// TIA Portal project "SocketConnection_Active" (V15.1)

(* hardware
DEVICE "S71500/ET200MP station_1"  S7-1500 station
   slot 0: "Rail_0"  Rack  6ES7 590-1***0-0AA0
   slot 1: "PLC_1"  CPU 1516-3 PN/DP  6ES7 516-3AN00-0AB0  V1.8
      slot 3: "CPU display_1"  6ES7591-1BA00-0AA0
DEVICE "S7-1200 station_1"  S7-1200 Station
   slot 0: "Rack_0"  S7-1200 Rack  Rack  V1.0
   slot 1: "PLC_2"  CPU 1212FC DC/DC/DC  6ES7 212-1AF40-0XB0  V4.2
*)

// ===== PLC "PLC_1"  CPU 1516-3 PN/DP =====

VAR_GLOBAL   // PLC tag table "Default tag table"
   "TCON_REQ" AT %M0.0 : Bool;
   "TSEND_REQ" AT %M0.1 : Bool;
   "Tag_3" AT %M0.2 : Bool;
   "Tag_4" AT %M0.3 : Bool;
   "TCON_DONE" AT %M0.4 : Bool;
   "TCON_BUSY" AT %M0.5 : Bool;
   "TCON_ERROR" AT %M0.6 : Bool;
   "TSEND_DONE" AT %M1.0 : Bool;
   "TSEND_ERROR" AT %M1.1 : Bool;
   "TSEND_BUSY" AT %M1.2 : Bool;
   "TRCV_NDR" AT %M1.3 : Bool;
   "TRCV_BUSY" AT %M1.4 : Bool;
   "TRCV_ERROR" AT %M1.5 : Bool;
   "Tag_14" AT %M1.6 : Bool;
   "TCON_DONE_PLS" AT %M1.7 : Bool;
   "TCON_DONE_COUNT" AT %MW100 : Int;
   "TSEND_DONE_PLS" AT %M2.0 : Bool;
   "TSEND_DONE_COUNT" AT %MW102 : Int;
   "Tag_19" AT %M3.1 : Bool;
   "Tag_20" AT %M5.0 : Bool;
   "Tag_21" AT %M3.3 : Bool;
   "CONNECT_RST" AT %M0.7 : Bool;
END_VAR

DATA_BLOCK "FB_TCPIP_Active_DB"   // DB6
{ S7_Optimized_Access := 'TRUE' }
VERSION : 0.1
// stored: InstanceOfName FB_TCPIP_Active
"FB_TCPIP_Active"
BEGIN
END_DATA_BLOCK

DATA_BLOCK "MyData"   // DB10
{ S7_Optimized_Access := 'FALSE' }
VERSION : 0.1
   VAR
      send_data : Array[1000..1719] of UInt;
      rcv_data : Array[0..9] of Byte;
   END_VAR
BEGIN
END_DATA_BLOCK

// folder: System blocks/Program resources

DATA_BLOCK "PLC_1_Connection_DB"   // DB2
{ S7_Optimized_Access := 'TRUE' }
AUTHOR : SIMATIC
FAMILY : MC7Plus
NAME : TC_IP_v4
VERSION : 1.0
// stored: InstanceOfName TCON_IP_v4
"TCON_IP_v4"
BEGIN
   ID := 1;
   InterfaceId := 64;
   LocalPort := 4000;
   RemotePort := 4000;
   ActiveEstablished := true;
   RemoteAddress.ADDR[1] := 192;
   RemoteAddress.ADDR[2] := 168;
   RemoteAddress.ADDR[4] := 251;
END_DATA_BLOCK

// folder: (top level)

FUNCTION_BLOCK "FB_TCPIP_Active"   // FB1, LAD
{ S7_Optimized_Access := 'TRUE' }
VERSION : 0.1
   VAR_INPUT
      REQ : Array[0..15] of Bool;
   END_VAR
   VAR
      TCON : TCON;
      TSEND : TSEND;
      TRCV : TRCV;
      TDISCON : TDISCON;
      pls : Array[0..15] of Bool;
      COUNT : Array[0..15] of Int;
   END_VAR
   VAR_TEMP   // added for the SCL form of the ladder/FBD networks
      _w1 : Bool;
      _w2 : Bool;
   END_VAR
   // // REQ[0] : TCON
   // // REQ[1] : TSEND
   // // REQ[2] : TDISCON
BEGIN

REGION Network 2: TON
END_REGION

REGION Network 3: ..Req
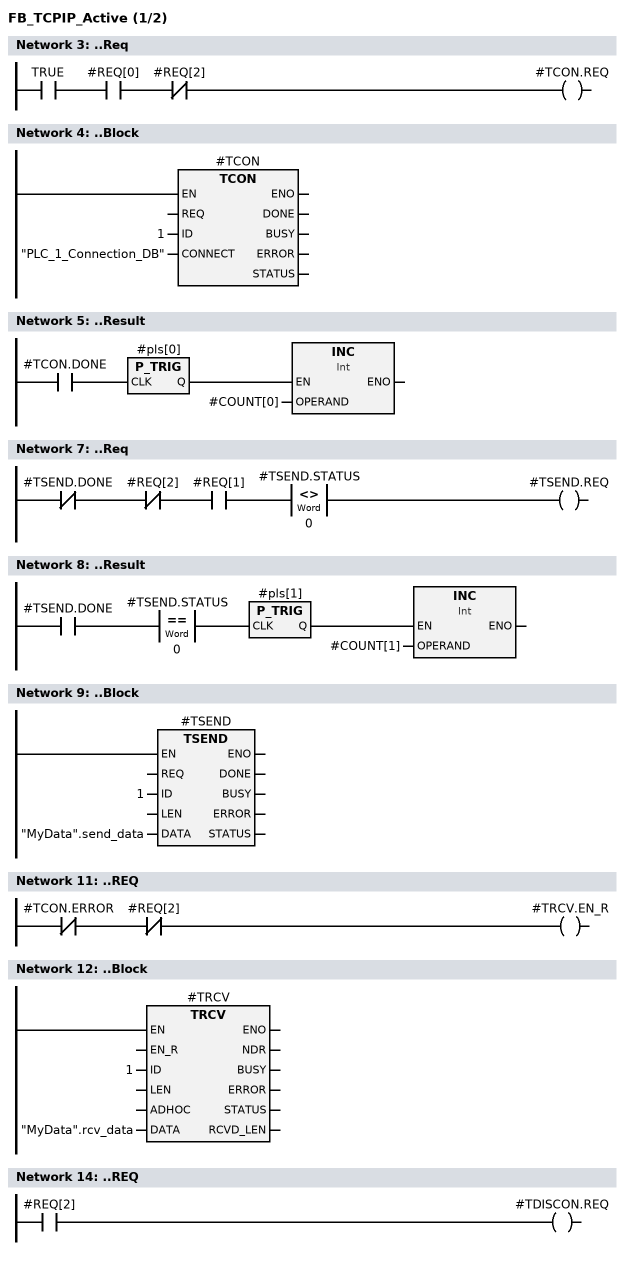
   RUNG wire#powerrail
      Contact( TRUE )
      Contact( #REQ[0] )
      I_Contact( #REQ[2] )
      Coil( #TCON.REQ )
   END_RUNG
   // the same network as SCL:
   #TCON.REQ := TRUE AND #REQ[0] AND NOT #REQ[2];
END_REGION

REGION Network 4: ..Block
   #TCON(ID := 1, CONNECT := "PLC_1_Connection_DB");   // TCON
END_REGION

REGION Network 5: ..Result
   RUNG wire#powerrail
      Contact( #TCON.DONE )
      P_Trig( #pls[0] )
      { S7_Templates := "DestType := Int" } Inc( #COUNT[0] )
   END_RUNG
   // the same network as SCL:
   #_w1 := #TCON.DONE AND NOT #pls[0];   // rising edge
   #pls[0] := #TCON.DONE;
   IF #_w1 THEN #COUNT[0] := #COUNT[0] + 1; END_IF;
END_REGION

REGION Network 6: TSEND
END_REGION

REGION Network 7: ..Req
   RUNG wire#powerrail
      I_Contact( #TSEND.DONE )
      I_Contact( #REQ[2] )
      Contact( #REQ[1] )
      { S7_Templates := "SrcType := Word" } NE_Contact(in1 := #TSEND.STATUS, in2 := 0)
      Coil( #TSEND.REQ )
   END_RUNG
   // the same network as SCL:
   #TSEND.REQ := NOT #TSEND.DONE AND NOT #REQ[2] AND #REQ[1] AND (#TSEND.STATUS <> 0);
END_REGION

REGION Network 8: ..Result
   RUNG wire#powerrail
      Contact( #TSEND.DONE )
      { S7_Templates := "SrcType := Word" } EQ_Contact(in1 := #TSEND.STATUS, in2 := 0)
      P_Trig( #pls[1] )
      { S7_Templates := "DestType := Int" } Inc( #COUNT[1] )
   END_RUNG
   // the same network as SCL:
   #_w1 := #TSEND.DONE AND (#TSEND.STATUS = 0);
   #_w2 := #_w1 AND NOT #pls[1];   // rising edge
   #pls[1] := #_w1;
   IF #_w2 THEN #COUNT[1] := #COUNT[1] + 1; END_IF;
END_REGION

REGION Network 9: ..Block
   #TSEND(ID := 1, DATA := "MyData".send_data);   // TSEND
END_REGION

REGION Network 10: TRCV
END_REGION

REGION Network 11: ..REQ
   RUNG wire#powerrail
      I_Contact( #TCON.ERROR )
      I_Contact( #REQ[2] )
      Coil( #TRCV.EN_R )
   END_RUNG
   // the same network as SCL:
   #TRCV.EN_R := NOT #TCON.ERROR AND NOT #REQ[2];
END_REGION

REGION Network 12: ..Block
   #TRCV(ID := 1, DATA := "MyData".rcv_data);   // TRCV
END_REGION

REGION Network 13: TDISCON
END_REGION

REGION Network 14: ..REQ
   RUNG wire#powerrail
      Contact( #REQ[2] )
      Coil( #TDISCON.REQ )
   END_RUNG
   // the same network as SCL:
   #TDISCON.REQ := #REQ[2];
END_REGION

REGION Network 15: ..Block
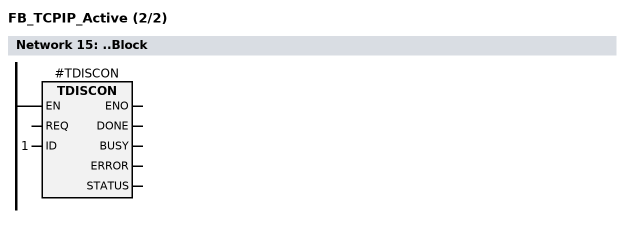
   #TDISCON(ID := 1);   // TDISCON
END_REGION
END_FUNCTION_BLOCK

FUNCTION "Backup" : Void   // FC1, LAD
{ S7_Optimized_Access := 'TRUE' }
VERSION : 0.1
   VAR_TEMP   // added for the SCL form of the ladder/FBD networks
      _w1 : Bool;
   END_VAR
BEGIN

REGION Network 2
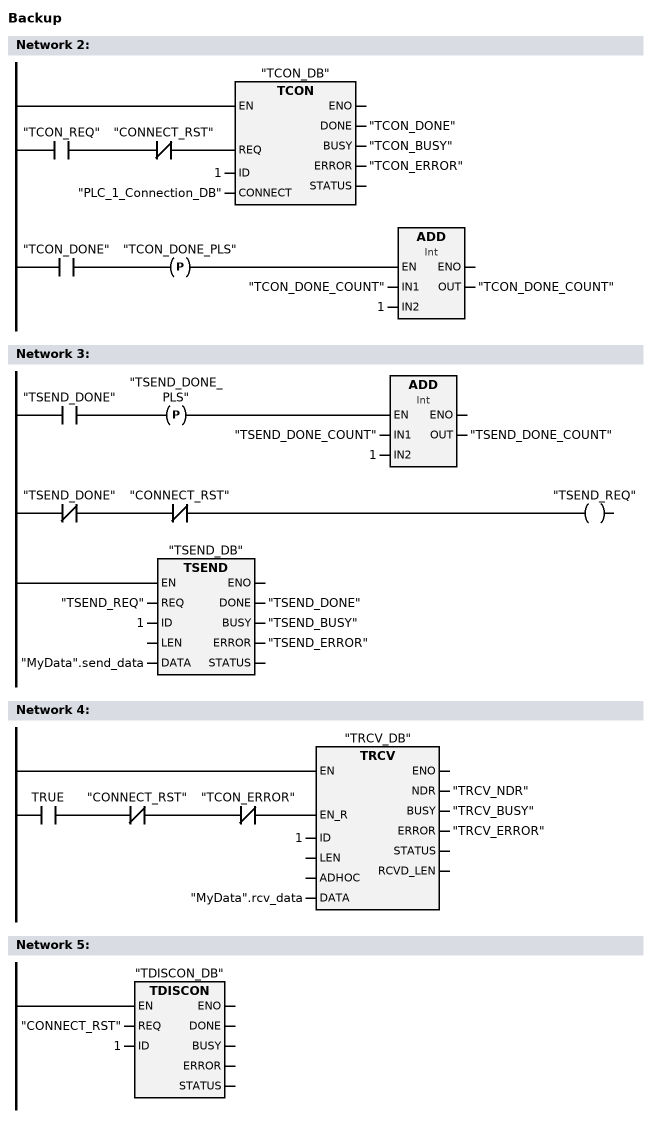
   "TCON_DB"(REQ := "TCON_REQ" AND NOT "CONNECT_RST",   // TCON
             ID := 1,
             CONNECT := "PLC_1_Connection_DB",
             DONE => "TCON_DONE",
             BUSY => "TCON_BUSY",
             ERROR => "TCON_ERROR");
   #_w1 := "TCON_DONE" AND NOT "TCON_DONE_PLS";   // rising edge
   "TCON_DONE_PLS" := "TCON_DONE";
   IF #_w1 THEN "TCON_DONE_COUNT" := "TCON_DONE_COUNT" + 1; END_IF;
END_REGION

REGION Network 3
   #_w1 := "TSEND_DONE" AND NOT "TSEND_DONE_PLS";   // rising edge
   "TSEND_DONE_PLS" := "TSEND_DONE";
   IF #_w1 THEN "TSEND_DONE_COUNT" := "TSEND_DONE_COUNT" + 1; END_IF;
   "TSEND_REQ" := NOT "TSEND_DONE" AND NOT "CONNECT_RST";
   "TSEND_DB"(REQ := "TSEND_REQ",   // TSEND
              ID := 1,
              DATA := "MyData".send_data,
              DONE => "TSEND_DONE",
              BUSY => "TSEND_BUSY",
              ERROR => "TSEND_ERROR");
END_REGION

REGION Network 4
   "TRCV_DB"(EN_R := TRUE AND NOT "CONNECT_RST" AND NOT "TCON_ERROR",   // TRCV
             ID := 1,
             DATA := "MyData".rcv_data,
             NDR => "TRCV_NDR",
             BUSY => "TRCV_BUSY",
             ERROR => "TRCV_ERROR");
END_REGION

REGION Network 5
   "TDISCON_DB"(REQ := "CONNECT_RST", ID := 1);   // TDISCON
END_REGION
END_FUNCTION

ORGANIZATION_BLOCK "Main"   // OB1, LAD, ProgramCycle
TITLE = "Main Program Sweep (Cycle)"
{ S7_Optimized_Access := 'TRUE' }
VERSION : 0.1
   VAR_INPUT
      Initial_Call : Bool;   // Initial call of this OB
      Remanence : Bool;   // =True, if remanent data are available
   END_VAR
   VAR_TEMP
      REQ : Array[0..15] of Bool;
   END_VAR
BEGIN

REGION Network 1
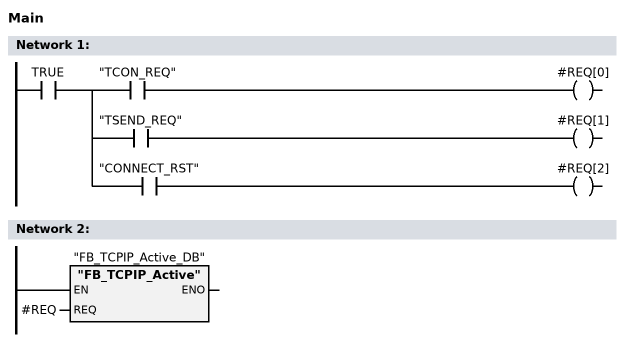
   RUNG wire#powerrail
      Contact( TRUE )
      wire#w1
      Contact( "TCON_REQ" )
      Coil( #REQ[0] )
   END_RUNG
   RUNG wire#w1
      Contact( "TSEND_REQ" )
      Coil( #REQ[1] )
   END_RUNG
   RUNG wire#w1
      Contact( "CONNECT_RST" )
      Coil( #REQ[2] )
   END_RUNG
   // the same network as SCL:
   #REQ[0] := TRUE AND "TCON_REQ";
   #REQ[1] := TRUE AND "TSEND_REQ";
   #REQ[2] := TRUE AND "CONNECT_RST";
END_REGION

REGION Network 2
   RUNG wire#powerrail
      "FB_TCPIP_Active_DB"(REQ := #REQ)
   END_RUNG
   // the same network as SCL:
   "FB_TCPIP_Active_DB"(REQ := #REQ);   // "FB_TCPIP_Active"
END_REGION
END_ORGANIZATION_BLOCK

// ===== PLC "PLC_2"  CPU 1212FC DC/DC/DC =====

VAR_GLOBAL   // PLC tag table "Default tag table"
   "TCON_REQ" AT %M0.0 : Bool;
   "TSEND_REQ" AT %M0.1 : Bool;
   "Tag_3" AT %M0.2 : Bool;
   "Tag_4" AT %M0.3 : Bool;
   "TCON_DONE" AT %M0.4 : Bool;
   "TCON_BUSY" AT %M0.5 : Bool;
   "TCON_ERROR" AT %M0.6 : Bool;
   "TSEND_DONE" AT %M1.0 : Bool;
   "TSEND_ERROR" AT %M1.1 : Bool;
   "TSEND_BUSY" AT %M1.2 : Bool;
   "TRCV_NDR" AT %M1.3 : Bool;
   "TRCV_BUSY" AT %M1.4 : Bool;
   "TRCV_ERROR" AT %M1.5 : Bool;
   "Tag_14" AT %M1.6 : Bool;
   "TCON_DONE_PLS" AT %M1.7 : Bool;
   "TCON_DONE_COUNT" AT %MW100 : Int;
   "TSEND_DONE_PLS" AT %M2.0 : Bool;
   "TSEND_DONE_COUNT" AT %MW102 : Int;
   "Tag_19" AT %M3.1 : Bool;
   "Tag_20" AT %M5.0 : Bool;
   "Tag_21" AT %M3.3 : Bool;
   "CONNECT_RST" AT %M0.7 : Bool;
   "Tag_1" AT %M4.0 : Bool;
END_VAR

DATA_BLOCK "MyData"   // DB10
{ S7_Optimized_Access := 'FALSE' }
VERSION : 0.1
   VAR
      send_data : Array[1000..1719] of UInt;
      rcv_data : Array[0..9] of Byte;
   END_VAR
BEGIN
END_DATA_BLOCK

// folder: System blocks/Program resources

DATA_BLOCK "PLC_1_Connection_DB"   // DB2
{ S7_Optimized_Access := 'TRUE' }
AUTHOR : SIMATIC
FAMILY : MC7Plus
NAME : TC_IP_v4
VERSION : 1.0
// stored: InstanceOfName TCON_IP_v4
"TCON_IP_v4"
BEGIN
   ID := 1;
   InterfaceId := 64;
   LocalPort := 4000;
   RemotePort := 4000;
   ActiveEstablished := true;
   RemoteAddress.ADDR[1] := 192;
   RemoteAddress.ADDR[2] := 168;
   RemoteAddress.ADDR[4] := 251;
END_DATA_BLOCK

// folder: (top level)

ORGANIZATION_BLOCK "Main"   // OB1, LAD, ProgramCycle
TITLE = "Main Program Sweep (Cycle)"
{ S7_Optimized_Access := 'TRUE' }
VERSION : 0.1
   VAR_INPUT
      Initial_Call : Bool;   // Initial call of this OB
      Remanence : Bool;   // =True, if remanent data are available
   END_VAR
   VAR_TEMP   // added for the SCL form of the ladder/FBD networks
      _w1 : Bool;
   END_VAR
BEGIN

REGION Network 2
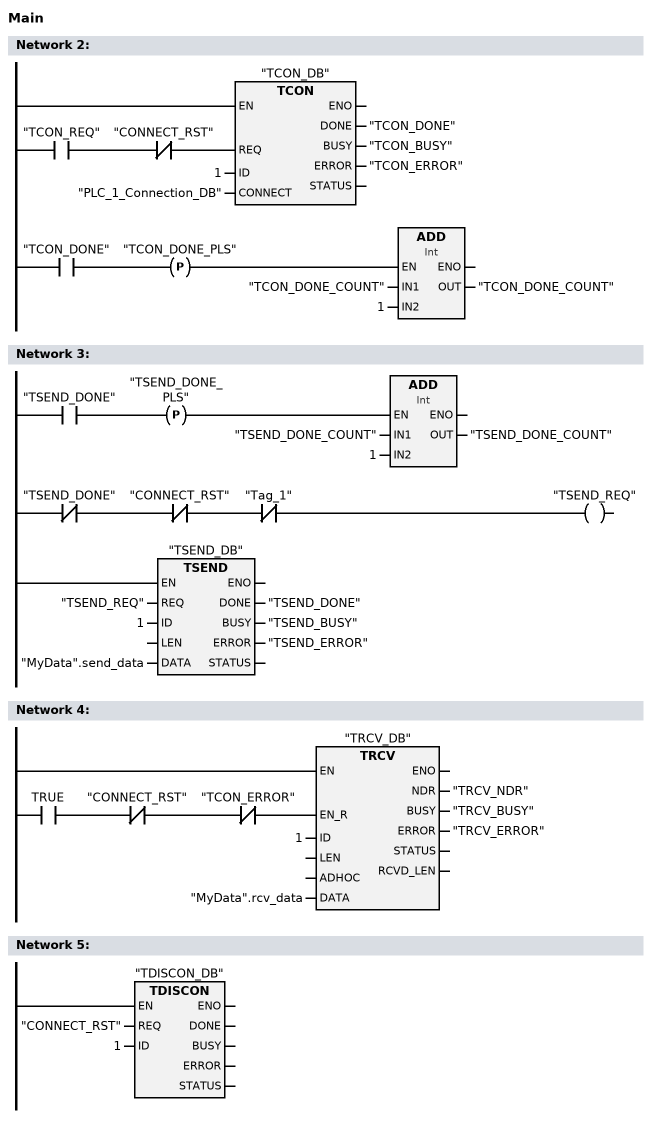
   "TCON_DB"(REQ := "TCON_REQ" AND NOT "CONNECT_RST",   // TCON
             ID := 1,
             CONNECT := "PLC_1_Connection_DB",
             DONE => "TCON_DONE",
             BUSY => "TCON_BUSY",
             ERROR => "TCON_ERROR");
   #_w1 := "TCON_DONE" AND NOT "TCON_DONE_PLS";   // rising edge
   "TCON_DONE_PLS" := "TCON_DONE";
   IF #_w1 THEN "TCON_DONE_COUNT" := "TCON_DONE_COUNT" + 1; END_IF;
END_REGION

REGION Network 3
   #_w1 := "TSEND_DONE" AND NOT "TSEND_DONE_PLS";   // rising edge
   "TSEND_DONE_PLS" := "TSEND_DONE";
   IF #_w1 THEN "TSEND_DONE_COUNT" := "TSEND_DONE_COUNT" + 1; END_IF;
   "TSEND_REQ" := NOT "TSEND_DONE" AND NOT "CONNECT_RST" AND NOT "Tag_1";
   "TSEND_DB"(REQ := "TSEND_REQ",   // TSEND
              ID := 1,
              DATA := "MyData".send_data,
              DONE => "TSEND_DONE",
              BUSY => "TSEND_BUSY",
              ERROR => "TSEND_ERROR");
END_REGION

REGION Network 4
   "TRCV_DB"(EN_R := TRUE AND NOT "CONNECT_RST" AND NOT "TCON_ERROR",   // TRCV
             ID := 1,
             DATA := "MyData".rcv_data,
             NDR => "TRCV_NDR",
             BUSY => "TRCV_BUSY",
             ERROR => "TRCV_ERROR");
END_REGION

REGION Network 5
   "TDISCON_DB"(REQ := "CONNECT_RST", ID := 1);   // TDISCON
END_REGION
END_ORGANIZATION_BLOCK